ABB RAPID module: AssemblerPosition.mod

MODULE AssemblerPosition
    CONST orient VERTICAL := [0.55931,-0.38758,0.51841,0.51789];

    CONST robtarget PICKUP := [ [172.4, 320.7, 315.0],  VERTICAL, [0,0,-1,1], [9E9,9E9,9E9,9E9,9E9,9E9] ];
    CONST robtarget SAFEPOSITION := [ [-115.5, 258.3, 400],  VERTICAL, [0,0,-1,1], [9E9,9E9,9E9,9E9,9E9,9E9] ];
    CONST robtarget DROP := [ [-100.9, 591.6, 250], VERTICAL, [0,0,-1,1], [9E9,9E9,9E9,9E9,9E9,9E9] ];

    CONST robtarget TABLETPOS1 := [ [149.8, 236.8, 331.5], VERTICAL, [0,0,-1,1], [9E9,9E9,9E9,9E9,9E9,9E9] ];
    CONST robtarget TABLETPOS2 := [ [211.8,236.8, 331.5], VERTICAL, [0,0,-1,1], [9E9,9E9,9E9,9E9,9E9,9E9] ];
    CONST robtarget TABLETPOS3 := [ [149.8, 279.7, 331.5],VERTICAL, [0,0,-1,1], [9E9,9E9,9E9,9E9,9E9,9E9] ];
    CONST robtarget TABLETPOS4 := [ [211.8, 279.7, 331.5], VERTICAL, [0,0,-1,1], [9E9,9E9,9E9,9E9,9E9,9E9] ];
    CONST robtarget TABLETPOS5 := [ [149.8, 364, 331.5], VERTICAL, [0,0,-1,1], [9E9,9E9,9E9,9E9,9E9,9E9] ];
    CONST robtarget TABLETPOS6 := [ [211.8, 364,331.5], VERTICAL, [0,0,-1,1], [9E9,9E9,9E9,9E9,9E9,9E9] ];
    CONST robtarget TABLETPOS7 := [ [149.8, 407.4, 331.5], VERTICAL, [0,0,-1,1], [9E9,9E9,9E9,9E9,9E9,9E9] ];
    CONST robtarget TABLETPOS8 := [ [211.8,407.4,331.5], VERTICAL, [0,0,-1,1], [9E9,9E9,9E9,9E9,9E9,9E9] ];
ENDMODULE
